(* IEC 61131-3 sources: MpAxisSample/axis01, 3 files *)

(* ---- Variables.var ---- *)
VAR
	interface : MpAxisInterfaceType;
END_VAR

(* ---- Init.st ---- *)
PROGRAM _INIT

	(* change following 3 lines for a new axis *)
	adrAxis01 := ADR(interface); //change "adrAxis01"
	interface.MpAxisBasic_0.MpLink := ADR(gAxisBasic01); //change "gAxisBasic01"
	interface.MpAxisBasic_0.Axis := ADR(gAxis01); //change "gAxis01"

END_PROGRAM

(* ---- Main.st ---- *)
PROGRAM _CYCLIC

	interface.MpAxisBasic_0.Enable := TRUE;
	interface.MpAxisBasic_0.Parameters := ADR(interface.parameters);
	interface.MpAxisBasic_0.Power := interface.power AND interface.MpAxisBasic_0.Info.ReadyToPowerOn;

	IF interface.MpAxisBasic_0.Info.PLCopenState = mpAXIS_ERRORSTOP OR interface.MpAxisBasic_0.Info.PLCopenState = mpAXIS_STOPPING THEN
		interface.MpAxisBasic_0.Update := FALSE;
		interface.MpAxisBasic_0.MoveVelocity := FALSE;
		interface.MpAxisBasic_0.MoveAbsolute := FALSE;
		interface.MpAxisBasic_0.MoveAdditive := FALSE;
		interface.MpAxisBasic_0.JogPositive := FALSE;
		interface.MpAxisBasic_0.JogNegative := FALSE;
		interface.MpAxisBasic_0.Autotune := FALSE;
	END_IF

	interface.MpAxisBasic_0();

	interface.MpAxisBasic_0.ErrorReset := FALSE;

	IF interface.MpAxisBasic_0.UpdateDone THEN
		interface.MpAxisBasic_0.Update := FALSE;
	END_IF

	IF interface.MpAxisBasic_0.InPosition THEN
		interface.MpAxisBasic_0.MoveAbsolute := FALSE;
		interface.MpAxisBasic_0.MoveAdditive := FALSE;
	END_IF

	IF interface.MpAxisBasic_0.TuningDone THEN
		interface.MpAxisBasic_0.Autotune := FALSE;
	END_IF

	interface.MpAxisBasic_0.Stop := FALSE;

END_PROGRAM

PROGRAM _EXIT

	interface.MpAxisBasic_0(Enable := FALSE);

END_PROGRAM
